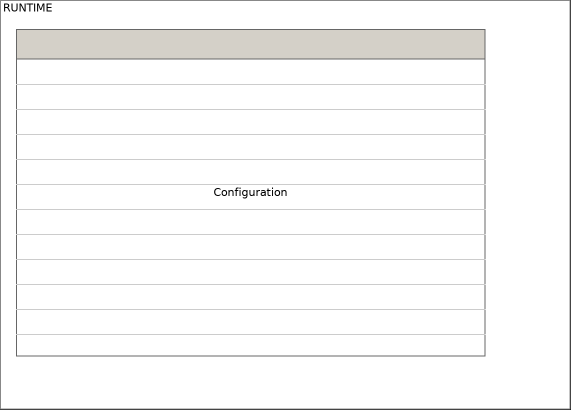
VISUALIZATION VI_XTSStationsRuntimeVisu  // 571x410
VAR_IN_OUT
	xts : XTS_System;
END_VAR
VAR
	stTableStruct : ARRAY [1..25] OF stTableStructx10;
END_VAR
    Rectangle (0,0 571x410), "RUNTIME"
    Table (16,29 469x327), "Configuration", data array: stTableStruct
        p3854506369: xts.stCfg.stStationsCfg[INDEX].sName
        p1892666644: xts.stCfg.stStationsCfg[INDEX].bEnableManualAck
        p338671338: xts.stCfg.stStationsCfg[INDEX].bManualAck
        p2170511999: xts.aStations[INDEX].fbMoversFIFO.nMovers
        p3723444502: xts.stCfg.stStationsCfg[INDEX].lrStopPosition[3]
        p1218418051: xts.stCfg.stStationsCfg[INDEX].lrProcessingTime
        p746581629: xts.stCfg.stStationsCfg[INDEX].uiNumStopPositions
        p3104783080: xts.stCfg.stStationsCfg[INDEX].lrTravelTime
        p7306298: xts.stCfg.stStationsCfg[INDEX].lrEndPosition
        p2685023577: stTableStruct.b1
        p511219082: Manual Ack
        p3312258591: stTableStruct.b2
        p1791247317: stTableStruct.b3
        p4092479075: Movers Waiting
        p262371475: stTableStruct.b4
        p2237128397: Stop Position 3
        p4008173056: stTableStruct.b5
        p505689113: Process Time
        p2340480326: stTableStruct.b6
        p1757482276: Stop Positions
        p606709900: stTableStruct.b7
        p4088588272: Travel Time
        p1095668682: stTableStruct.b8
        p2243050616: Extra Cfg.
        p1037165547: stTableStruct.b9
        p516019884: End Position
        p1488378029: stTableStruct.b10
        Columns.Column.[3].Template: xts.aStations[INDEX].bWaitingMovers
        Columns.Column.[6].Template: OnMouseClick: write the text variable via Default, min 1, max 3
        Columns.Column.[4].Template: OnMouseClick: write the text variable via Default
        Columns.Column.[5].Template: OnMouseClick: write the text variable via Default
        Columns.Column.[2].Template: tap xts.stCfg.stStationsCfg[INDEX].bManualAck
        Columns.Column.[0].Template: OnMouseClick: write the text variable via Default
        Columns.Column.[7].Template: OnMouseClick: write the text variable via Default
        Columns.Column.[9].Template: OnMouseClick: write the text variable via Default
        Columns.Column.[1].Template: toggle xts.stCfg.stStationsCfg[INDEX].bEnableManualAck
END_VISUALIZATION

(* stored: Version 1.1.0.1, ProductVersion 3.1.4024.11
   Visu VI_XTSStationsRuntimeVisu: Id {f9e20e03-8613-4e3e-8212-6b9c477a923d} *)
